DATA_BLOCK "pump_start_stop_DB4"
{ S7_Optimized_Access := 'TRUE' }
VERSION : 0.1
NON_RETAIN
"pump_start_stop"

BEGIN

END_DATA_BLOCK

